(* PLC project , OpenPLC Project OpenPLC Editor v3 *)

PROGRAM Main

PROGRAM Main
VAR
    Rising : R_EDGE;
END_VAR
Rising(CLK := TRUE);
END_PROGRAM
END_PROGRAM

PROGRAM LegacySfc

PROGRAM LegacySfc
END_PROGRAM
END_PROGRAM
